PROGRAM A22
VAR_IN_OUT
	sectionCC : CardboardEx;
	
	bundlesQueue : ARRAY[0..CONSTS.maxQueue] OF Bundle;
	bundlesBypass : ARRAY[0..CONSTS.maxQueue] OF BOOL;
END_VAR
VAR
	robot3, robot4 : RobotA22;
	
	benderA22Left : FoldingMachine;
	
	skidA22Left, skidA22Right : SkidMagazine;
	magazineA22Left, magazineA22Right : SkidMagazine;
	
	wrapperA22 : WrapMachine;
	overhead : STRING;
	
	horizontalDriveA22Left, horizontalDriveA22Right : ServoNC := (
		limitSensorDefaultState := TRUE);
		
	verticalDriveA22Left, verticalDriveA22Right : ClearLinkMC := (
		limitSensorDefaultState := TRUE, 
		homingDirectionOut := TRUE, //outwards (up)
		minPosition := (26*5 * 25.4),
		displacementPerRotation := 5,
		unitsPerPulse := 800); //800 counts = 1 rotation
		
	insertionA22Left, insertionA22Right : Insertion;

	pistonA22Bottom : SimplePiston;
	
	(*
	each insertion suction array has 3 pads
	[1] - top/bottom
	[2] - corner
	[3] - side
	*)
	suctionA22TopLeft : ARRAY[1..3] OF SuctionPad;
	suctionA22TopRight : ARRAY[1..3] OF SuctionPad;
	suctionA22BottomLeft : ARRAY[1..3] OF SuctionPad; 
	suctionA22BottomRight : ARRAY[1..3] OF SuctionPad;
	
	suctionA22Bottom : ARRAY[1..2] OF SuctionPad;
END_VAR
VAR //data arrays to be passed into material holder FBs - do not access directly
	skidHmiA22Left, skidHmiA22Right AT %M* : ARRAY[1...Cardboard.size-1] OF MaterialSlot;
	magazineHmiA22Left, magazineHmiA22Right AT %M* : ARRAY[1..CornerGuard.size-1] OF MaterialSlot;
END_VAR
VAR //other
	conveyorsCC : ARRAY[1..3] OF POINTER TO ConveyorSC;
END_VAR

callHardware();

setupHardware();

runModules();

callHardware();

METHOD PRIVATE callHardware : BOOL
skidA22Left(slots := skidHmiA22Left);
skidA22Right(slots := skidHmiA22Right);
magazineA22Left(slots := magazineHmiA22Left);
magazineA22Right(slots := magazineHmiA22Right);

wrapperA22(extSafety := robot3.wrapSafetyIn AND robot4.wrapSafetyIn);

verticalDriveA22Left(
	bEnable:= , 
	pulse=> , 
	brakeRelease=> , 
	enable=> , 
	A=> , 
	B=> , 
	clear=> );
verticalDriveA22Right(
	bEnable:= , 
	pulse=> , 
	brakeRelease=> , 
	enable=> , 
	A=> , 
	B=> , 
	clear=> );

horizontalDriveA22Left(bEnable:= TRUE, ready=> , position=> , velocity=> );
horizontalDriveA22Right(bEnable:= TRUE, ready=> , position=> , velocity=> );

insertionA22Left(
	slider:= verticalDriveA22Left, 
	screw:= horizontalDriveA22Left, 
	contact=> , 
	active=> , 
	error=> , 
	home=> , 
	homingComplete=> , 
	sliderPos=> );
	
insertionA22Right(
	slider:= verticalDriveA22Right, 
	screw:= horizontalDriveA22Right, 
	contact=> , 
	active=> , 
	error=> , 
	home=> , 
	homingComplete=> , 
	sliderPos=> );
END_METHOD

METHOD PRIVATE runModules : BOOL
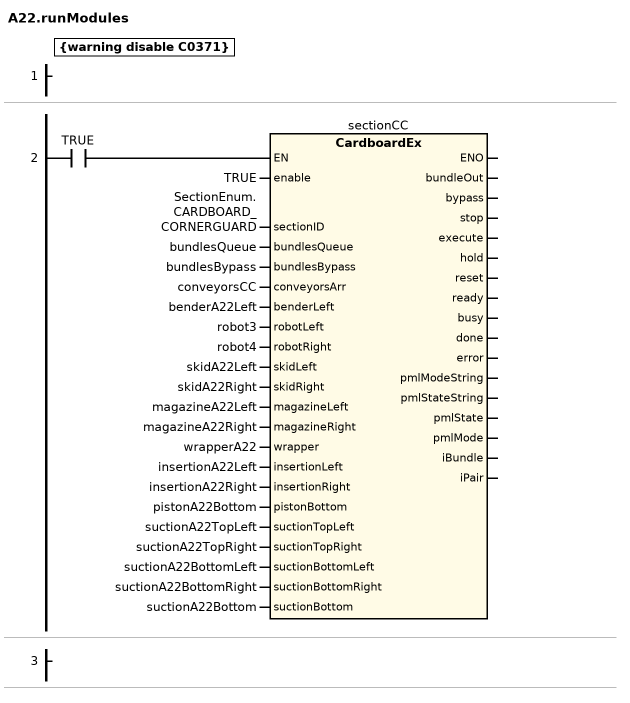
// NETWORK 1
// label: {warning disable C0371}

// NETWORK 2
sectionCC(
    enable := TRUE,
    sectionID := SectionEnum.CARDBOARD_CORNERGUARD,
    bundlesQueue := bundlesQueue,
    bundlesBypass := bundlesBypass,
    conveyorsArr := conveyorsCC,
    benderLeft := benderA22Left,
    robotLeft := robot3,
    robotRight := robot4,
    skidLeft := skidA22Left,
    skidRight := skidA22Right,
    magazineLeft := magazineA22Left,
    magazineRight := magazineA22Right,
    wrapper := wrapperA22,
    insertionLeft := insertionA22Left,
    insertionRight := insertionA22Right,
    pistonBottom := pistonA22Bottom,
    suctionTopLeft := suctionA22TopLeft,
    suctionTopRight := suctionA22TopRight,
    suctionBottomLeft := suctionA22BottomLeft,
    suctionBottomRight := suctionA22BottomRight,
    suctionBottom := suctionA22Bottom); // CardboardEx

// NETWORK 3
END_METHOD

METHOD PRIVATE setupHardware : BOOL
VAR
	iCornerGuardSlot : CornerGuard;
	iCardboardSlot : Cardboard;
	i : INT;
END_VAR
FOR iCornerGuardSlot:=1 TO WoodBunk.size-1 BY 1 DO //init wood bunk magazine slots
	magazineA22Left.setSlot(i := iCornerGuardSlot, material := TO_STRING(iCornerGuardSlot), error => );
	magazineA22Right.setSlot(i := iCornerGuardSlot, material := TO_STRING(iCornerGuardSlot), error => );
END_FOR

//--------------------------------------------------

FOR iCardboardSlot:=1 TO Chipboard.size-1 BY 1 DO //init chipboard skid slots
	skidA22Left.setSlot(i := iCardboardSlot, material := TO_STRING(iCardboardSlot), error => );
	skidA22Right.setSlot(i := iCardboardSlot, material := TO_STRING(iCardboardSlot), error => );
END_FOR

//--------------------------------------------------

FOR i:=1 TO CONSTS.maxQueue BY 1 DO //get corner guard magazine + cardboard skid availability from robot3 and robot4
	{warning disable C0195}
	skidA22Left.setOccupancy( i := i, occupancy := IntegerBitAccess(robot3.inputs[4], i-1) );
	skidA22Right.setOccupancy( i := i, occupancy := IntegerBitAccess(robot4.inputs[4], i-1) );

	magazineA22Left.setOccupancy( i := i, occupancy := IntegerBitAccess(robot4.inputs[3], i-1) );
	magazineA22Right.setOccupancy( i := i, occupancy := IntegerBitAccess(robot4.inputs[3], i-1) );
END_FOR

//--------------------------------------------------

conveyorsCC[1] := ADR(ConveyorSyncUnit.A22_SC_C15);
conveyorsCC[2] := ADR(ConveyorSyncUnit.A22_LSC_C16);
conveyorsCC[3] := ADR(ConveyorSyncUnit.A22_LSC_C17);
END_METHOD

END_PROGRAM

(* stored: Version 1.1.0.1, ProductVersion 3.1.4024.11
   POU A22: Id {1b16486c-3037-4854-af07-df0c4a7cb5bc}, SpecialFunc None
   Method callHardware: Id {f4d985bb-fe7d-48e1-9a81-baebf0e31a92}
   Method runModules: Id {610921f0-756a-4d32-a8a7-bd908cf51f55}
   Method setupHardware: Id {665ab571-9ad5-4fd6-97d1-c6a60483f8fb} *)
